{attribute addProperty BoxType "EK1122-0000-0018"}
{attribute addProperty Id "Beckhoff_ELM3xxxsub_EK1100EK1100_179A0949162"}
{attribute addProperty CRC "1386471739"}
{attribute addProperty SizeInBites "16"}
{attribute addProperty SizeInBytes "2"}
TYPE Beckhoff_ELM3xxxEK1122_52A3E13B EXTENDS EK1122_179A0949 :
STRUCT
	{attribute addProperty Name "Beckhoff_ELM3xxxsub_EK1100"}
	Beckhoff_ELM3xxxsub_EK1100 : EK1100_179A0949;
END_STRUCT
END_TYPE

(* stored: Version 1.2.0.0, ProductVersion 3.1.4024.9
   DUT Beckhoff_ELM3xxxEK1122_52A3E13B: Id {891e541a-dbd1-4f3d-836a-8d06df3d12b4} *)
